ScreenModuleEditorView "Row_Material" 600x40
   Rectangle "Border" at 0,0 size 600x40
      Visibility <- "interface.background_visible"
      Appearance <- "interface.background_animate"
   TextField "TF R0 C0" at 5,5 size 360x35; Text 'MOLYBDENUM'
      Visibility <- "interface.cell_0_visible"
      Appearance <- "interface.cell_0_animate"
   IOField "IOF R0 C1" at 370,5 size 225x35; FormatPattern 9999999
      on OnFinishInput: SetBit("interface.cell_1_input_finished")
      Visibility <- "interface.cell_1_visible"
      ObjectEnable <- "interface.cell_1_enable"
      Appearance <- "interface.cell_1_animate"
      on Activate: SetBit("interface.cell_1_active")
      on Deactivate: ResetBit("interface.cell_1_active")
*)

(* ===== HMI "HMI_RT_1" =====

ScreenModuleEditorView "Row_Material_Label" 600x40
   Rectangle "Border" at 0,0 size 600x40
      Visibility <- "interface.background_visible"
      Appearance <- "interface.background_animate"
   TextField "TF R0 C0" at 5,5 size 360x35; Text 'MATERIAL'
      Visibility <- "interface.cell_0_visible"
      Appearance <- "interface.cell_0_animate"
   TextField "TF R0 C1" at 370,5 size 225x35; Text 'BAGS'
      Visibility <- "interface.cell_1_visible"
      Appearance <- "interface.cell_1_animate"
*)

(* ===== HMI "HMI_RT_1" =====
system functions are stored by id; their names below are inferred from use

ScreenModuleEditorView "Row_Custom" 600x40
   Rectangle "Border" at 0,0 size 600x40
      Visibility <- "interface.background_visible"
      Appearance <- "interface.background_animate"
   IOField "IOF R0 C0" at 5,5 size 360x35; FormatPattern ???????????????
      on OnFinishInput: SetBit("interface.cell_0_input_finished")
      ObjectEnable <- "interface.cell_0_enable"
      Visibility <- "interface.cell_0_visible"
      Appearance <- "interface.cell_0_animate"
      on Activate: SetBit("interface.cell_0_activate")
      on Deactivate: ResetBit("interface.cell_0_activate")
   IOField "IOF R0 C1" at 370,5 size 225x35; FormatPattern 9999999
      on OnFinishInput: SetBit("interface.cell_1_input_finished")
      Visibility <- "interface.cell_1_visible"
      ObjectEnable <- "interface.cell_1_enable"
      Appearance <- "interface.cell_0_animate"
      on Activate: SetBit("interface.cell_1_activate")
      on Deactivate: ResetBit("interface.cell_1_activate")
*)

(* ===== HMI "HMI_RT_1" =====
system functions are stored by id; their names below are inferred from use

ScreenModuleEditorView "Row_Wire" 600x65
   Rectangle "Border" at 0,0 size 600x65
      Visibility <- "interface.background_visible"
      Appearance <- "interface.background_animate"
   TextField "TF R0 C0" at 5,5 size 360x60; Text 'CARBON WIRE'
      Visibility <- "interface.cell_0_visible"
      Appearance <- "interface.cell_0_animate"
   IOField "IOF R0 C1" at 370,5 size 225x60; FormatPattern ???????
      on Deactivate: ResetBit("interface.cell_1_active")
      on OnFinishInput: SetBit("interface.cell_1_input_finished")
      on Activate: SetBit("interface.cell_1_active")
      Visibility <- "interface.cell_1_visible"
      ObjectEnable <- "interface.cell_1_enable"
      Appearance <- "interface.cell_1_animate"
      ProcessValue <- "interface.cell_1_value"
*)

(* ===== HMI "HMI_RT_1" =====
system functions are stored by id; their names below are inferred from use

ScreenModuleEditorView "Row_Material" 600x40
   Rectangle "Border" at 0,0 size 600x40
      Visibility <- "interface.background_visible"
      Appearance <- "interface.background_animate"
   TextField "TF R0 C0" at 5,5 size 360x35; Text 'MOLYBDENUM'
      Visibility <- "interface.cell_0_visible"
      Appearance <- "interface.cell_0_animate"
   IOField "IOF R0 C1" at 370,5 size 225x35; FormatPattern ?????????
      on OnFinishInput: SetBit("interface.cell_1_input_finished")
      on Deactivate: ResetBit("interface.cell_1_active")
      on Activate: SetBit("interface.cell_1_active")
      Appearance <- "interface.cell_1_animate"
      Visibility <- "interface.cell_1_visible"
      ObjectEnable <- "interface.cell_1_enable"
      ProcessValue <- "interface.cell_1_value"
*)

(* ===== HMI "HMI_RT_1" =====
system functions are stored by id; their names below are inferred from use

ScreenModuleEditorView "Row_Custom" 600x40
   Rectangle "Border" at 0,0 size 600x40
      Visibility <- "interface.background_visible"
      Appearance <- "interface.background_animate"
   IOField "IOF R0 C0" at 5,5 size 360x35; FormatPattern ???????????????
      on OnFinishInput: SetBit("interface.cell_0_input_finished")
      on Deactivate: ResetBit("interface.cell_0_activate")
      on Activate: SetBit("interface.cell_0_activate")
      Appearance <- "interface.cell_0_animate"
      Visibility <- "interface.cell_0_visible"
      ObjectEnable <- "interface.cell_0_enable"
      ProcessValue <- "interface.cell_0_value"
   IOField "IOF R0 C1" at 370,5 size 225x35; FormatPattern ?????????
      on OnFinishInput: SetBit("interface.cell_1_input_finished")
      on Deactivate: ResetBit("interface.cell_1_activate")
      on Activate: SetBit("interface.cell_1_activate")
      Appearance <- "interface.cell_0_animate"
      Visibility <- "interface.cell_1_visible"
      ObjectEnable <- "interface.cell_1_enable"
      ProcessValue <- "interface.cell_1_value"
*)

(* ===== HMI "HMI_RT_1" =====
system functions are stored by id; their names below are inferred from use

ScreenModuleEditorView "Row_Custom" 600x40
   Rectangle "Border" at 0,0 size 600x40
      Visibility <- "interface.background_visible"
      Appearance <- "interface.background_animate"
   IOField "IOF R0 C0" at 5,5 size 360x35; FormatPattern ???????????????
      on Deactivate: ResetBit("interface.cell_0_activate")
      on OnFinishInput: SetBit("interface.cell_0_input_finished")
      on Activate: SetBit("interface.cell_0_activate")
      ProcessValue <- "interface.cell_0_value"
      Visibility <- "interface.cell_0_visible"
      Appearance <- "interface.cell_0_animate"
      ObjectEnable <- "interface.cell_0_enable"
   IOField "IOF R0 C1" at 370,5 size 225x35; FormatPattern ?????????
      on Deactivate: ResetBit("interface.cell_1_activate")
      on OnFinishInput: SetBit("interface.cell_1_input_finished")
      on Activate: SetBit("interface.cell_1_activate")
      ProcessValue <- "interface.cell_1_value"
      Visibility <- "interface.cell_1_visible"
      ObjectEnable <- "interface.cell_1_enable"
      Appearance <- "interface.cell_1_animate"
*)